FUNCTION F_ECat_OK : BOOL
VAR_INPUT
	State : WORD;	// State from Ethercat module/device
END_VAR
VAR
END_VAR

// Check etherCAT state OK
F_ECat_OK := (State AND 16#0008) = 8;
IF bTestMode THEN
	F_ECat_OK := TRUE;
END_IF

END_FUNCTION

(* stored: Version 1.1.0.1, ProductVersion 3.1.4024.2
   POU F_ECat_OK: Id {3258f906-cbd3-45ce-9a4c-bc675666a334}, SpecialFunc None *)
